// TIA Portal project "Projekt1" (V15.1)

(* hardware
DEVICE "S7-1200-Station_1"  S7-1200 Station
   slot 0: "Baugruppenträger_0"  S7-1200 Rack  Rack  V1.0
   slot 1: "PLC_1"  CPU 1215C AC/DC/Rly  6ES7 215-1BG40-0XB0  V4.2
*)

// ===== PLC "PLC_1"  CPU 1215C AC/DC/Rly =====

VAR_GLOBAL   // PLC tag table "Standard-Variablentabelle"
   "System_Byte" AT %MB444 : Byte;
   "FirstScan" AT %M444.0 : Bool;
   "DiagStatusUpdate" AT %M444.1 : Bool;
   "AlwaysTRUE" AT %M444.2 : Bool;
   "AlwaysFALSE" AT %M444.3 : Bool;
   "Clock_Byte" AT %MB333 : Byte;
   "Clock_10Hz" AT %M333.0 : Bool;
   "Clock_5Hz" AT %M333.1 : Bool;
   "Clock_2.5Hz" AT %M333.2 : Bool;
   "Clock_2Hz" AT %M333.3 : Bool;
   "Clock_1.25Hz" AT %M333.4 : Bool;
   "Clock_1Hz" AT %M333.5 : Bool;
   "Clock_0.625Hz" AT %M333.6 : Bool;
   "Clock_0.5Hz" AT %M333.7 : Bool;
END_VAR

VAR_GLOBAL   // PLC tag table "Variablentabelle_1"
   "Start-Taster" AT %I0.0 : Bool;
   "Stop-Taster" AT %I0.1 : Bool;
   "Motorschutzschalter" AT %I0.2 : Bool;
   "Motorschütz" AT %Q0.0 : Bool;
   "Störungslampe" AT %Q0.1 : Bool;
END_VAR

DATA_BLOCK "Datenbaustein_Motorschaltung"   // DB1
{ S7_Optimized_Access := 'TRUE' }
VERSION : 0.1
   VAR
      WebStart : Bool;
      WebStop : Bool := true;
   END_VAR
BEGIN
END_DATA_BLOCK

FUNCTION "Motorsteuerung mit Selbsthaltung" : Void   // FC1, FBD
{ S7_Optimized_Access := 'TRUE' }
VERSION : 0.1
BEGIN

REGION Network 1
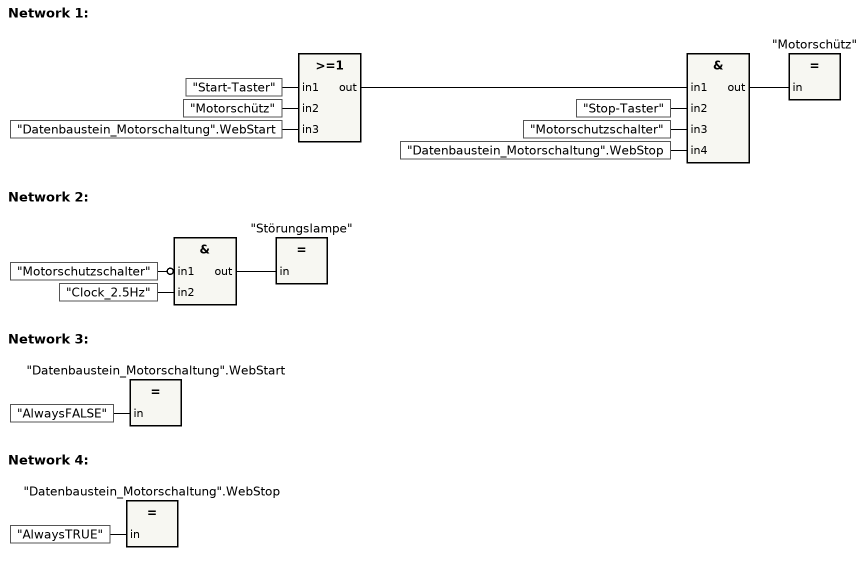
   "Motorschütz" := ("Start-Taster" OR "Motorschütz" OR "Datenbaustein_Motorschaltung".WebStart) AND "Stop-Taster" AND "Motorschutzschalter" AND "Datenbaustein_Motorschaltung".WebStop;
END_REGION

REGION Network 2
   "Störungslampe" := NOT "Motorschutzschalter" AND "Clock_2.5Hz";
END_REGION

REGION Network 3
   "Datenbaustein_Motorschaltung".WebStart := "AlwaysFALSE";
END_REGION

REGION Network 4
   "Datenbaustein_Motorschaltung".WebStop := "AlwaysTRUE";
END_REGION
END_FUNCTION

ORGANIZATION_BLOCK "Main"   // OB1, LAD, ProgramCycle
TITLE = "Main Program Sweep (Cycle)"
{ S7_Optimized_Access := 'TRUE' }
VERSION : 0.1
   VAR_INPUT
      Initial_Call : Bool;   // Initial call of this OB
      Remanence : Bool;   // =True, if remanent data are available
   END_VAR
BEGIN

REGION Network 1
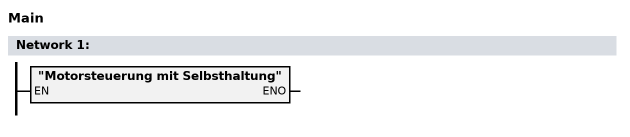
   RUNG wire#powerrail
      "Motorsteuerung mit Selbsthaltung"()
   END_RUNG
   // the same network as SCL:
   "Motorsteuerung mit Selbsthaltung"();
END_REGION
END_ORGANIZATION_BLOCK